// TIA Portal V19 export
FUNCTION "PB_CIP FILLER" : Void   // FC90, STL
TITLE = Pb - CIP filling mashine
{ S7_Optimized_Access := 'TRUE' }
NAME : PBLYECIP
VERSION : 0.0
// Comment
// stored: AutoNumber false
   VAR_TEMP
      alarmbit : Int;
   END_VAR
BEGIN

NETWORK
TITLE = 
// Comment Flash K9 when filler ready for CIP
//       AN    I     32.2
      AN    "S0 CIP TANK";
      AN    "S0 CHAIN WASH";
      =     "LEDAssignment".K9_FLASH;  //"FLASH_K9_CIP_FIL"
      =     "M_CIP_FILLER_READY";
//      JC    B001

// **** This section has been added ... AFL
//      A     "Combi 512 is in use"       //512 INTERFACE IN USE
//      A     "FILLER_ENABLE"             //
//      R     "LEDAssignment".K9_FLASH    // "FLASH_K9_CIP_FIL"

// **** End ***************************************
//B001: NOP   0


NETWORK
TITLE = ALARM 51
// CIP Blocing
// 
//       A     I     32.2                  // FILLER CIP SIGNAL MISSING
//       A     "S0 FILLER"
//       JC    C001                        // STOP CIP 
// 
//  **** This section has been added ... AFL
//       A     "Combi 512 is in use"       //512 INTERFACE IN USE
//       AN    "FILLER_ENABLE"             // FILLER CIP SIGNAL MISSING
// 
//       A     "S0 FILLER"
//       JC    C001                        // STOP CIP 
//  **** End ***************************************
      AN    "LEDAssignment".K9_BUTTON;  // "PbK9CIPFILLER" // START/STOP CIP FILLER

      BEC;
      R     "LEDAssignment".K9_BUTTON;  //"PbK9CIPFILLER"


      A     "S0 FILLER";
      JC    C001;  // STOP CIP

// **** This section has been added ... AFL
//      A     "Combi 512 is in use"       //512 INTERFACE IN USE
//      AN    "FILLER_ENABLE"
//      S     "A51-FILLER NOT READY"      // FILLER NOT RADY FOR CIP
//      BEC

// **** End ***************************************
      A     "S0 CIP TANK";
      S     "ProcessAndPbAlarms"."A"[14];  //A14_CipOnTankStared// CIP TANK STARTED
      L     14;
      JC    Alrm;

//      BEC
      O     "CHAIN_WASH";
      O     "S0 CHAIN WASH";
      S     "ProcessAndPbAlarms"."A"[15];  //A15_ChainWashSelected// CHAIN WASH SELECTED
      L     15;
      JC    Alrm;

//      BEC
      AN    "CIP_PROG_1";
      AN    "CIP_PROG_2";
      AN    "CIP_PROG_3";
      S     "ProcessAndPbAlarms"."A"[16];  //A16_NoCipProgramSelected// NO PROGRAM SELECTED
      L     16;
      JC    Alrm;

//      BEC
      AN    "PA0572_Air";
      S     "ProcessAndPbAlarms"."A"[3];  //A03_NoInstrumentAir// no instrument air
      L     3;
      JC    Alrm;

//      BEC
      AN    "PA0561_Steam";
      S     "ProcessAndPbAlarms"."A"[4];  //A04_NoSteam// no steam
      L     4;
      JC    Alrm;

//      BEC
      S     "S0 FILLER";
      S     "LEDAssignment".K9_FLASH;  //"FLASH_K9_CIP_FIL"
      S     "LEDAssignment".K9_LIGHT;  //"LIGHT_K9_CIP_FIL"
      BEU;

C001: R     "S0 FILLER";
      R     "LEDAssignment".K9_FLASH;  //"FLASH_K9_CIP_FIL"
      R     "LEDAssignment".K9_LIGHT;  // "LIGHT_K9_CIP_FIL"
      R     "AutoTT0172/IP0157";
      R     "MM0139";
      R     "MY0114";  // drain
      R     "MY0115";
      R     "MY0116";
      R     "MY0117";
      R     "MY0119";
      R     "CONTROL CIP TANK";
      R     "S.T.01.REQUEST LYE";
      R     "S.T.01.REQUEST ACID";
      R     "M_RINSE_READY";
      R     "M_CAUSTIC_READY";
      R     "M_ACID_READY";
      R     "RINSE_READY";
      R     "CAUSTIC_READY";
      R     "ACID_READY";
      BEU;



NETWORK
TITLE = Blockings alarm text
// Blockings alarm
Alrm: NOP   1;
      T     #alarmbit;
      CALL  "Set_Pop_Up_Blocking"
      ( alarmTextNum := #alarmbit
      );  // start blockings text


END_FUNCTION
